{attribute 'qualified_only'}
{attribute 'strict'}
TYPE E_HygState :
(
 	ST_IDLE := 0,
    ST_WAIT_FILL,
    ST_DOSE_PERLITE,
    ST_MIX_1,
    ST_DOSE_CAO,
    ST_MIX_2,
    ST_OPEN_GATE,
    ST_DISCHARGE,
    ST_CLOSE_GATE,
    ST_DONE,
    ST_ALARM
);
END_TYPE

(* stored: Version 1.1.0.1, ProductVersion 3.1.4024.15
   DUT E_HygState: Id {1514d64d-bd7c-4272-8a70-54a048644641} *)
